// TIA Portal V19 export
VAR_GLOBAL   // PLC tag table "LB114"
   LB114_Rollformer_Lp_Bwd AT %Q118.1 : Bool;   // 330SH2
   LB114_Rollformer_Lp_Fwd AT %Q118.0 : Bool;   // 330SH1
   LB114_Rollformer_Pb_Bwd AT %I121.2 : Bool;   // 330SH2
   LB114_Rollformer_Pb_Fwd AT %I121.1 : Bool;   // 330SH1
   LB114_Straightener_Lp_Bwd AT %Q118.3 : Bool;   // 330SH4
   LB114_Straightener_Lp_Fwd AT %Q118.2 : Bool;   // 330SH3
   LB114_Straightener_Pb_Bwd AT %I121.4 : Bool;   // 330SH4
   LB114_Straightener_Pb_Fwd AT %I121.3 : Bool;   // 330SH3
   LB114_Button_L AT %I1072.0 : Bool;   // 105DI0 - 202SB1
   LB114_Button_R AT %I1072.4 : Bool;   // 105DI4 - 202SB2
END_VAR
